// TIA Portal V21 export
DATA_BLOCK "MV3000LineAnimationDb"   // DB801
// stored: AutoNumber false, InstanceOfName MV3000LineAnimation, InstanceOfType FB
"MV3000LineAnimation"
   // VAR_INPUT
   //    AlwaysTrue : Bool;
   //    AlwaysFalse : Bool;
   //    SecPulse : Bool;
   //    "Spare 1" : Bool;
   //    "Spare 2" : Bool;
   //    "Spare 3" : Bool;
   //    "Spare 4" : Bool;
   //    "Spare 5" : Bool;
   // END_VAR
   // VAR
   //    "Node 1" : "LineAnimationFb";
   //    "Node 2" : "LineAnimationFb";
   //    "Node 3" : "LineAnimationFb";
   //    "Node 4" : "LineAnimationFb";
   //    "Node 5" : "LineAnimationFb";
   //    "Node 6" : "LineAnimationFb";
   //    "Node 7" { S7_SetPoint := 'True'} : "LineAnimationFb";
   //    "Node 8" { S7_SetPoint := 'True'} : "LineAnimationFb";
   //    "Node 9" { S7_SetPoint := 'True'} : "LineAnimationFb";
   //    "Node 10" { S7_SetPoint := 'True'} : "LineAnimationFb";
   //    "Node 11" { S7_SetPoint := 'True'} : "LineAnimationFb";
   //    "Node 12" { S7_SetPoint := 'True'} : "LineAnimationFb";
   //    "Node 13" { S7_SetPoint := 'True'} : "LineAnimationFb";
   //    "Node 14" { S7_SetPoint := 'True'} : "LineAnimationFb";
   //    "Node 15" { S7_SetPoint := 'True'} : "LineAnimationFb";
   //    "Node 16" { S7_SetPoint := 'True'} : "LineAnimationFb";
   //    "Node 17" { S7_SetPoint := 'True'} : "LineAnimationFb";
   //    "Node 18" { S7_SetPoint := 'True'} : "LineAnimationFb";
   //    "Node 19" { S7_SetPoint := 'True'} : "LineAnimationFb";
   //    "Node 20" { S7_SetPoint := 'True'} : "LineAnimationFb";
   //    "Node 21" { S7_SetPoint := 'True'} : "LineAnimationFb";
   //    "Node 22" { S7_SetPoint := 'True'} : "LineAnimationFb";
   //    "Node 23" { S7_SetPoint := 'True'} : "LineAnimationFb";
   //    "Node 24" { S7_SetPoint := 'True'} : "LineAnimationFb";
   //    "Node 25" { S7_SetPoint := 'True'} : "LineAnimationFb";
   //    "Node 26" { S7_SetPoint := 'True'} : "LineAnimationFb";
   //    "Node 27" { S7_SetPoint := 'True'} : "LineAnimationFb";
   //    "Node 28" { S7_SetPoint := 'True'} : "LineAnimationFb";
   //    "Node 29" { S7_SetPoint := 'True'} : "LineAnimationFb";
   //    "Node 30" { S7_SetPoint := 'True'} : "LineAnimationFb";
   //    Node31 { S7_SetPoint := 'True'} : "LineAnimationFb";
   //    Node32 { S7_SetPoint := 'True'} : "LineAnimationFb";
   //    Node33 { S7_SetPoint := 'True'} : "LineAnimationFb";
   //    Node34 { S7_SetPoint := 'True'} : "LineAnimationFb";
   // END_VAR
BEGIN
END_DATA_BLOCK
